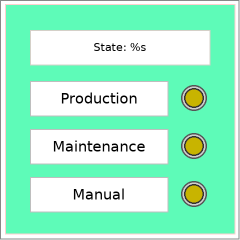
VISUALIZATION V_Module  // 240x240
VAR_IN_OUT
	HMI : ST_PackMLBaseModule_HMI;
END_VAR
    RoundedRectangle (5,4 230x230)
    Textfield (30,30 180x35), "State: %s", text variable: HMI.Status.State
    Lamp1 (179,83 30x30), variable: HMI.Status.Mode = E_PMLUnitMode.ePMLUnitMode_Production, style: Lamp-Lamp1-Yellow
    Lamp1 (179,131 30x30), variable: HMI.Status.Mode = E_PMLUnitMode.ePMLUnitMode_Maintenance, style: Lamp-Lamp1-Yellow
    Lamp1 (179,179 30x30), variable: HMI.Status.Mode = E_PMLUnitMode.ePMLUnitMode_Manual, style: Lamp-Lamp1-Yellow
    RoundedRectangle (30,81 138x35), "Production"
        OnMouseClick: execute { HMI.Command.Mode := E_PMLUnitMode.ePMLUnitMode_Production; }
    RoundedRectangle (30,129 138x35), "Maintenance"
        OnMouseClick: execute { HMI.Command.Mode := E_PMLUnitMode.ePMLUnitMode_Maintenance; }
    RoundedRectangle (30,177 138x35), "Manual"
        OnMouseClick: execute { HMI.Command.Mode := E_PMLUnitMode.ePMLUnitMode_Manual; }
END_VISUALIZATION

(* stored: Version 1.1.0.1
   Visu V_Module: Id {ab5ca517-81c1-49dd-92aa-b6c97677d45a} *)
